PROGRAM MAIN
VAR
	fbGenerateTimeData_TEST	:	GenerateTimeData_TEST;
	fbHelperFunctions_TEST: ConvertAnyToString_TEST;
	testWrapper	:	TestWrapper_NET();
END_VAR

TcUnit.RUN();

testWrapper();

END_PROGRAM

(* stored: Version 1.1.0.1, ProductVersion 3.1.4024.4
   POU MAIN: Id {899b5391-5363-4fd8-835e-d1662fef51af}, SpecialFunc None *)
